(* IEC 61131-3 sources: codesys-build/examples/frame-assembly/src/transport/PRG_Transport, 1 file *)

(* ---- declaration.st ---- *)
PROGRAM PRG_Transport
VAR
	Conveyor : FB_Conveyor;
	ClampedSpeed : INT;
END_VAR
